// TIA Portal V19 export
FUNCTION_BLOCK "TYPIC_C106_IF_MVI"   // FB84, FBD
TITLE = TYPIC_C106_IF_MVI: Hoogspanningsverdeelbord
{ S7_Optimized_Access := 'TRUE' }
AUTHOR : OCOTECH
FAMILY : Typical
NAME : C106.702
// Logisch Object Besturing: C106.702
// 
// De interne functie Hoogspanningsverdeelbord verzorgt de bewaking van een oogspanningsverdeelbord.
// stored: MemoryReserve 10, SetENOAutomatically false
   VAR_INPUT
      EXT_AUT { ExternalAccessible := 'False'; ExternalVisible := 'False'; ExternalWritable := 'False'} : Bool;   // Externe (hoofd) beveiliging (1 = OK)
      EXT_HW { ExternalAccessible := 'False'; ExternalVisible := 'False'; ExternalWritable := 'False'} : Bool;   // Sturings hardware (PLC) bewaking (1 = OK)
      IN_PWR1 { ExternalAccessible := 'False'; ExternalVisible := 'False'; ExternalWritable := 'False'} : Real;   // Actief vermogen
      IN_PWR2 { ExternalAccessible := 'False'; ExternalVisible := 'False'; ExternalWritable := 'False'} : Real;   // Reactief vermogen
      IN_SPA1 { ExternalAccessible := 'False'; ExternalVisible := 'False'; ExternalWritable := 'False'} : Real;   // Lijnspanning 1
      IN_SPA2 { ExternalAccessible := 'False'; ExternalVisible := 'False'; ExternalWritable := 'False'} : Real;   // Lijnspanning 2
      IN_SPA3 { ExternalAccessible := 'False'; ExternalVisible := 'False'; ExternalWritable := 'False'} : Real;   // Lijnspanning 3
      IN_PSU_STO { ExternalAccessible := 'False'; ExternalVisible := 'False'; ExternalWritable := 'False'} : Bool;   // Storing door een fout op de UPS
      IN_PSU_AUT { ExternalAccessible := 'False'; ExternalVisible := 'False'; ExternalWritable := 'False'} : Bool;   // Verzamelalarm actief: de beveiliging van de hulpvoeding is getript
      IN_AUT_C106 { ExternalAccessible := 'False'; ExternalVisible := 'False'; ExternalWritable := 'False'} : Bool;   // Beveiligingen: serie geschakelde terugmelding (1 = OK)
   END_VAR
   VAR_OUTPUT
      VAR_IF_MVI { ExternalAccessible := 'False'; ExternalVisible := 'False'; ExternalWritable := 'False'} : "C106_VAR_IF_MVI_TYPIC";   // Struct met alle variabelen naar bovenliggende functies
   END_VAR
   VAR
      STO { ExternalWritable := 'False'} : Struct   // Storingen
         A001 : Bool;   // Beveiliging aangesproken
         A002 : Bool;   // Hoogspanningsverdeelbord in storing
         A003 : Bool;   // Algemene storing hoogspanningsverdeelbord
         A004 : Bool;   // Alarm door een fout op de UPS
         A005 : Bool;   // Verzamelalarm actief: de beveiliging van de hulpvoeding is getript
      END_STRUCT;
      VAR { ExternalWritable := 'False'} : Struct   // Variabelen
         PWR1 : Real;   // Geleverde actief vermogen per aggregaat
         PWR2 : Real;   // Geleverde reactief vermogen per aggregaat
         SPA1 : Real;   // Spanningsniveau lijn 1
         SPA2 : Real;   // Spanningsniveau lijn 2
         SPA3 : Real;   // Spanningsniveau lijn 3
         PSU_STO : Bool;   // Storing door een fout op de UPS
         PSU_AUT : Bool;   // Verzamelalarm actief: de beveiliging van de hulpvoeding is getript
         EXT_AUT { ExternalAccessible := 'False'; ExternalVisible := 'False'} : Bool;   // Externe (hoofd) beveiliging aangesproken
         EXT_HW { ExternalAccessible := 'False'; ExternalVisible := 'False'} : Bool;   // Sturings hardware (PLC) in storing
      END_STRUCT;
   END_VAR
BEGIN

REGION Network 1: START
END_REGION

REGION Network 2: +++ Verwerking meetwaarden en statussen +++
   // De meetwaarde en status wordt ontvangen vanuit de interne sturing.
END_REGION

REGION Network 3: +++ Storingen +++
   // Verwerken van de storingsmeldingen (inputs).
END_REGION

REGION Network 4: Storing A001: Beveiliging aangesproken
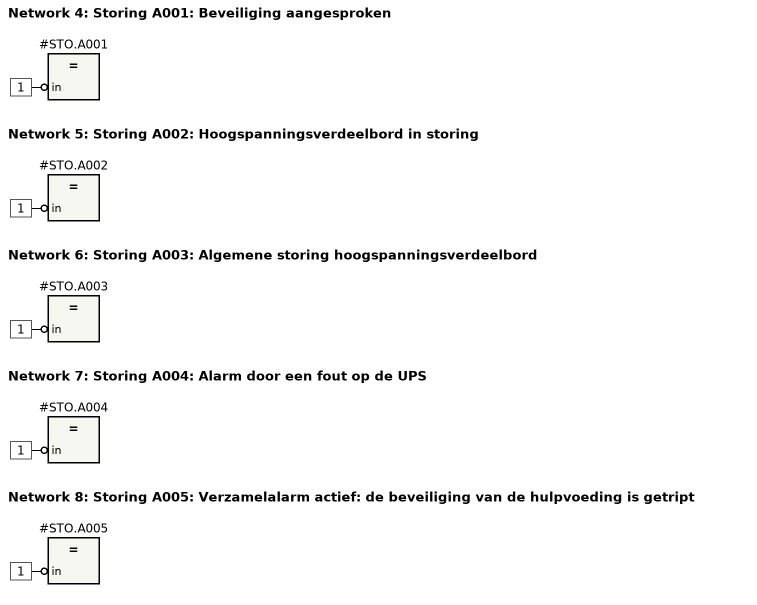
   #STO.A001 := NOT 1;
END_REGION

REGION Network 5: Storing A002: Hoogspanningsverdeelbord in storing
   #STO.A002 := NOT 1;
END_REGION

REGION Network 6: Storing A003: Algemene storing hoogspanningsverdeelbord
   #STO.A003 := NOT 1;
END_REGION

REGION Network 7: Storing A004: Alarm door een fout op de UPS
   #STO.A004 := NOT 1;
END_REGION

REGION Network 8: Storing A005: Verzamelalarm actief: de beveiliging van de hulpvoeding is getript
   #STO.A005 := NOT 1;
END_REGION

REGION Network 9 (SCL): EINDE
   // Variabelen van intern scada rakvlak naar outputs copieren
   #VAR_IF_MVI.PWR1 := #VAR.PWR1;
   #VAR_IF_MVI.PWR2 := #VAR.PWR2;
   #VAR_IF_MVI.SPA1 := #VAR.SPA1;
   #VAR_IF_MVI.SPA2 := #VAR.SPA2;
   #VAR_IF_MVI.SPA3 := #VAR.SPA3;
   #VAR_IF_MVI.PSU_STO := #VAR.PSU_STO;
   #VAR_IF_MVI.PSU_AUT := #VAR.PSU_AUT;
   #VAR_IF_MVI.EXT_AUT := #VAR.EXT_AUT;
   #VAR_IF_MVI.EXT_HW := #VAR.EXT_HW;
   #VAR_IF_MVI.STO := #STO;
END_REGION
END_FUNCTION_BLOCK
